PROGRAM Singulation_Control_1
VAR
	SortSingulation	:	FB_Singulation;
	RetryLimit		:	UINT := 1;
	ReleaseDist		:	UINT;
END_VAR

SortSingulation(
//	In_ConveyorRunning := Conveyors.P8005_VFD.IsRunning,
//	In_Grabber_1_Auto := Solenoids.GR8005_1_Status.Sts_EquipmentState.StsAuto,
//	In_Grabber_1_Extended := ProxSensors.In_PX_22741_Extended,
//	In_Grabber_1_Retracted := ProxSensors.In_PX_22721_Retracted,
//	In_Grabber_2_Auto := Solenoids.GR8005_2_Status.Sts_EquipmentState.StsAuto,
//	In_Grabber_2_Extended := ProxSensors.In_PX_23341_Extended,
//	In_Grabber_2_Retracted := ProxSensors.In_PX_23321_Retracted,
//	In_PinStop_Auto := Solenoids.PS8005_Status.Sts_EquipmentState.StsAuto,
//	In_PinStop_Extended := ProxSensors.In_PX_22541_Extended,
//	In_PinStop_Retracted := ProxSensors.In_PX_22521_Retracted,
	In_FaultReset := System.Cnvyr_Reset,
//	In_EncoderCount := GVL_IO.ENC_11321_Raw,
//	In_PE_GrabTrigger:= PhotoEyes.PE_22521.Out_OnFltrd, 
//	In_PE_ToteTrigger:= PhotoEyes.PE_22501.Out_OffFltrd, 
//	In_PE_ClearedTrigger:= PhotoEyes.PE_22621.Out_OffFltrd,
	Cfg_GappingDistance := ReleaseDist,
	Cfg_TimeOutTime:= T#5S,
	Cfg_RetryLimit:= RetryLimit, 
);

END_PROGRAM

(* stored: Version 1.1.0.1, ProductVersion 3.1.4024.4
   POU Singulation_Control_1: Id {29efa8a8-80d0-4e8c-b871-cc6beb136689}, SpecialFunc None *)
